Yaskawa INFORM job: BATMAN_2STR.JBI

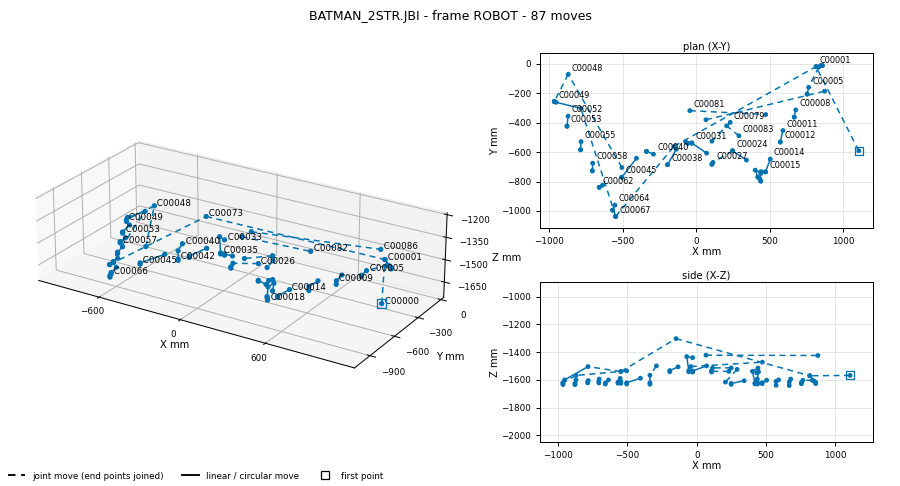
[picture p0: tool path of BATMAN_2STR.JBI in frame ROBOT, 87 of 158 moves have a stored position in this frame; points joined in program order, loops and branches not executed]
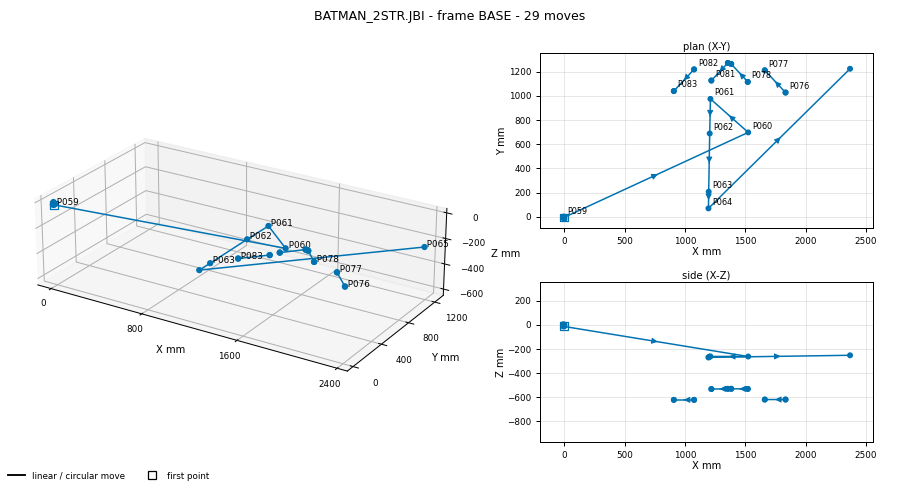
[picture p1: tool path of BATMAN_2STR.JBI in frame BASE, 29 of 158 moves have a stored position in this frame; points joined in program order, loops and branches not executed]
/JOB
//NAME BATMAN_2STR
///FOLDERNAME KRIS-SCIANA
//POS
///NPOS 87,87,0,38,0,0
///TOOL 0
///POSTYPE ROBOT
///RECTAN
///RCONF 0,0,0,0,0,0,0,0,0,0,0,0,0,0,0,0,0,0,0,0,0,0,0,0
C00000=1105.156,-590.615,-1567.354,6.0584,32.6468,147.4704
C00001=815.315,-18.001,-1569.939,-1.7381,27.7880,143.5527
C00002=857.710,-10.973,-1618.417,-1.7378,27.7886,143.5541
C00003=857.707,-10.971,-1626.567,-1.7382,27.7883,143.5526
C00004=833.675,-21.061,-1602.919,-1.7360,27.7873,143.5574
C00005=764.713,-159.460,-1602.917,-1.7360,27.7871,143.5577
C00006=754.333,-205.391,-1618.911,-1.7368,27.7882,143.5563
C00007=754.360,-205.381,-1627.221,-1.7390,27.7891,143.5536
C00008=676.929,-312.752,-1594.094,-1.7387,27.7900,143.5534
C00009=666.860,-361.337,-1616.296,-1.7391,27.7907,143.5606
C00010=666.607,-362.154,-1640.305,-1.7382,27.7861,143.5578
C00011=589.702,-453.220,-1599.704,-1.7386,27.7882,143.5565
C00012=571.550,-531.474,-1610.685,-1.7384,27.7889,143.5556
C00013=571.577,-531.526,-1638.417,-1.7371,27.7932,143.5506
C00014=503.343,-647.565,-1602.574,-1.7244,27.7369,143.5385
C00015=471.201,-734.222,-1620.126,-1.7395,27.7918,143.5502
C00016=471.196,-734.208,-1626.856,-1.7400,27.7912,143.5505
C00017=439.050,-796.935,-1621.095,-1.7408,27.7924,143.5517
C00018=439.049,-796.953,-1629.727,-1.7399,27.7928,143.5504
C00019=441.123,-742.830,-1514.057,-1.7418,27.7901,143.5526
C00020=401.170,-722.445,-1537.720,10.1454,37.8099,55.1563
C00021=419.273,-769.804,-1621.635,10.0244,37.5346,56.2633
C00022=419.267,-769.795,-1628.682,10.0249,37.5342,56.2644
C00023=341.517,-653.963,-1605.800,10.0246,37.5341,56.2657
C00024=247.787,-591.524,-1625.473,10.0271,37.5316,56.2731
C00025=247.794,-591.522,-1631.709,10.0263,37.5313,56.2715
C00026=247.796,-591.525,-1513.148,10.0256,37.5315,56.2705
C00027=113.704,-669.750,-1513.152,10.0280,37.5312,56.2733
C00028=106.856,-682.927,-1533.943,10.0224,37.5325,56.2697
C00029=106.874,-682.958,-1542.733,10.0189,37.5339,56.2663
C00030=70.694,-606.931,-1498.730,10.0200,37.5334,56.2633
C00031=-30.272,-538.287,-1535.198,10.0214,37.5337,56.2637
C00032=-30.275,-538.292,-1543.514,10.0219,37.5340,56.2653
C00033=-30.277,-538.270,-1439.519,10.0239,37.5323,56.2676
C00034=-72.212,-529.493,-1431.848,10.0246,37.5336,126.4601
C00035=-58.288,-539.735,-1534.232,10.0230,37.5329,126.4597
C00036=-58.298,-539.747,-1541.111,10.0251,37.5325,126.4632
C00037=-134.942,-579.910,-1505.733,10.0214,37.5335,126.4526
C00038=-194.951,-685.626,-1532.619,10.0192,37.5313,126.4507
C00039=-194.945,-685.631,-1541.099,10.0183,37.5324,126.4483
C00040=-291.274,-613.943,-1498.709,10.0193,37.5315,126.4500
C00041=-338.146,-594.905,-1566.079,10.0206,37.5306,126.4559
C00042=-338.153,-594.908,-1620.637,10.0213,37.5304,126.4568
C00043=-338.152,-594.897,-1631.211,10.0213,37.5296,126.4575
C00044=-406.496,-641.674,-1587.377,10.0204,37.5303,126.4602
C00045=-505.818,-770.602,-1620.991,10.0161,37.5294,126.4561
C00046=-505.822,-770.602,-1629.641,10.0170,37.5289,126.4582
C00047=-505.818,-704.683,-1534.604,10.0172,37.5293,126.4596
C00048=-870.558,-70.607,-1567.754,-5.5732,23.9550,-0.0620
C00049=-965.415,-255.754,-1620.582,-3.4263,30.0338,0.8210
C00050=-965.418,-255.752,-1622.018,-3.4258,30.0337,0.8220
C00051=-965.421,-255.747,-1633.054,-3.4254,30.0337,0.8221
C00052=-871.675,-355.111,-1600.349,-3.4260,30.0340,0.8216
C00053=-878.724,-423.891,-1625.207,-3.4243,30.0345,0.8253
C00054=-878.718,-423.902,-1634.168,-3.4261,30.0338,0.8213
C00055=-782.869,-528.764,-1604.816,-3.4248,30.0318,0.8156
C00056=-786.737,-583.960,-1612.292,-3.4246,30.0303,0.8183
C00057=-786.740,-583.966,-1621.129,-3.4247,30.0307,0.8203
C00058=-704.142,-675.428,-1593.875,-3.4274,30.0320,0.8194
C00059=-706.471,-727.273,-1611.725,-3.4351,30.0238,0.8165
C00060=-706.461,-727.277,-1621.357,-3.4355,30.0231,0.8168
C00061=-637.422,-825.106,-1600.424,-3.4351,30.0208,0.8167
C00062=-659.834,-839.485,-1622.110,-3.4334,30.0214,0.8205
C00063=-659.844,-839.500,-1629.778,-3.4344,30.0221,0.8200
C00064=-552.859,-959.979,-1588.724,-3.4350,30.0244,0.8136
C00065=-568.518,-994.720,-1614.958,-3.4362,30.0232,0.8143
C00066=-568.514,-994.724,-1623.430,-3.4363,30.0225,0.8125
C00067=-547.865,-1036.819,-1613.327,-3.4355,30.0239,0.8160
C00068=-547.869,-1036.811,-1624.522,-3.4350,30.0238,0.8135
C00069=-547.867,-1036.815,-1539.725,-3.4353,30.0236,0.8134
C00070=-784.559,-302.239,-1503.879,-3.4366,30.0265,0.8087
C00071=-953.024,-261.100,-1599.401,-3.4345,30.0250,0.8092
C00072=-547.867,-1036.815,-1539.725,-3.4353,30.0236,0.8134
C00073=-149.962,-559.854,-1302.120,-3.4346,30.0247,0.8146
C00074=815.315,-18.001,-1569.939,-1.7381,27.7880,143.5527
C00075=847.137,-11.115,-1608.986,-1.7371,27.7876,143.5542
C00076=432.100,-781.158,-1548.511,-1.7395,27.7865,143.5518
C00077=445.125,-733.631,-1540.567,-2.7194,23.4640,36.3665
C00078=436.491,-734.622,-1593.359,-2.7195,23.4653,36.3724
C00079=231.186,-397.551,-1538.170,10.0369,37.5564,56.2933
C00080=106.565,-525.549,-1538.164,10.0364,37.5570,56.2931
C00081=-43.468,-317.794,-1503.609,10.0906,37.0928,60.8768
C00082=472.745,-344.262,-1471.900,21.7977,37.1280,159.9819
C00083=290.461,-488.573,-1524.026,10.0019,37.5312,126.4207
C00084=206.735,-421.024,-1615.254,10.0028,37.5295,126.4201
C00085=66.048,-379.716,-1421.439,10.0175,37.5426,126.4581
C00086=873.206,-185.580,-1423.876,-1.7383,27.7862,-167.3950
BC00000=938.923,1838.231,1681.523
BC00001=1421.588,1829.899,1010.263
BC00002=1421.588,1829.899,1010.263
BC00003=1421.588,1829.899,1010.263
BC00004=1421.581,1829.905,1010.257
BC00005=1421.581,1829.905,1010.257
BC00006=1421.581,1829.905,1010.257
BC00007=1421.581,1829.905,1010.257
BC00008=1421.581,1829.905,1010.257
BC00009=1421.581,1829.905,1010.257
BC00010=1421.581,1829.905,1010.257
BC00011=1421.581,1829.905,1010.257
BC00012=1421.581,1829.905,1010.257
BC00013=1421.581,1829.905,1010.257
BC00014=1421.581,1829.905,1010.257
BC00015=1421.581,1829.905,1010.257
BC00016=1421.581,1829.905,1010.257
BC00017=1421.581,1829.905,1010.257
BC00018=1421.581,1829.905,1010.257
BC00019=1421.581,1829.905,1010.254
BC00020=1421.581,1829.912,1010.248
BC00021=1414.141,1827.243,1016.162
BC00022=1414.141,1827.243,1016.162
BC00023=1414.141,1827.243,1016.162
BC00024=1414.141,1827.243,1016.162
BC00025=1414.141,1827.243,1016.162
BC00026=1414.141,1827.243,1016.162
BC00027=1414.141,1827.243,1016.162
BC00028=1414.141,1827.243,1016.162
BC00029=1414.141,1827.243,1016.162
BC00030=1414.141,1827.243,1016.162
BC00031=1414.141,1827.243,1016.162
BC00032=1414.141,1827.243,1016.162
BC00033=1414.141,1827.243,1016.162
BC00034=1414.141,1827.243,1016.162
BC00035=1414.141,1827.243,1016.162
BC00036=1414.141,1827.243,1016.162
BC00037=1414.141,1827.243,1016.162
BC00038=1414.141,1827.243,1016.162
BC00039=1414.141,1827.243,1016.162
BC00040=1414.141,1827.243,1016.162
BC00041=1414.141,1827.243,1016.162
BC00042=1414.141,1827.243,1016.162
BC00043=1414.141,1827.243,1016.162
BC00044=1414.141,1827.243,1016.162
BC00045=1414.141,1827.243,1016.162
BC00046=1414.141,1827.243,1016.162
BC00047=1414.141,1827.243,1016.162
BC00048=1421.581,1829.905,1010.254
BC00049=1421.581,2077.513,1010.254
BC00050=1421.581,2077.513,1010.254
BC00051=1421.581,2077.513,1010.254
BC00052=1421.581,2077.513,1010.248
BC00053=1421.581,2077.513,1010.248
BC00054=1421.581,2077.513,1010.248
BC00055=1421.581,2077.513,1010.248
BC00056=1421.581,2077.513,1010.248
BC00057=1421.581,2077.513,1010.248
BC00058=1421.581,2077.513,1010.248
BC00059=1421.581,2077.507,1010.244
BC00060=1421.581,2077.507,1010.244
BC00061=1421.581,2077.507,1010.244
BC00062=1421.581,2077.507,1010.244
BC00063=1421.581,2077.507,1010.244
BC00064=1421.581,2077.507,1010.244
BC00065=1421.581,2077.507,1010.244
BC00066=1421.581,2077.507,1010.244
BC00067=1421.581,2077.507,1010.244
BC00068=1421.581,2077.507,1010.244
BC00069=1421.581,2077.507,1010.244
BC00070=1421.581,2077.507,1010.244
BC00071=1421.581,2077.507,1010.244
BC00072=1421.581,2077.507,1010.244
BC00073=1421.581,2077.507,1010.244
BC00074=1421.588,1829.899,1010.263
BC00075=1421.588,1829.899,1010.263
BC00076=1421.588,1829.899,1010.263
BC00077=1421.588,1829.899,1010.263
BC00078=1421.588,1829.899,1010.263
BC00079=1436.938,1677.545,1031.627
BC00080=1436.938,1677.545,1031.627
BC00081=1441.270,1634.546,1037.657
BC00082=838.758,1634.546,1037.657
BC00083=842.369,1626.975,1038.719
BC00084=842.369,1626.975,1038.719
BC00085=842.362,1626.982,1038.713
BC00086=845.778,2972.171,1682.637
///POSTYPE BASE
P00059=-2.448,-6.714,-12.718,0.0000,0.0000,0.0000
P00060=1524.284,698.404,-261.973,-0.4635,36.8346,-1.2388
P00061=1211.499,975.999,-261.374,0.5148,35.2356,175.5099
P00062=1205.574,689.500,-262.704,0.5159,35.2461,175.5270
P00063=1197.217,207.358,-268.729,0.4863,35.2395,175.4586
P00064=1195.199,68.975,-269.171,0.5092,35.2366,175.4908
P00065=2367.684,1225.356,-251.745,0.6375,35.5356,-175.5535
P00070=2.449,-18.318,2.615,0.0000,0.0000,0.0000
P00071=-2.048,-0.034,-9.092,0.0000,0.0000,0.0000
P00072=-1.595,-0.049,-6.373,0.0000,0.0000,0.0000
P00073=-8.474,-10.331,-11.894,0.0000,0.0000,0.0000
P00074=1.731,-3.007,-10.460,0.0000,0.0000,0.0000
///RCONF 0,1,0,0,0,0,0,0,0,0,0,0,0,0,0,0,0,0,0,0,0,0,0,0
P00075=-9.634,0.014,4.922,0.0000,0.0000,0.0000
///RCONF 0,0,0,0,0,0,0,0,0,0,0,0,0,0,0,0,0,0,0,0,0,0,0,0
P00076=1833.500,1028.615,-618.215,10.0256,37.5190,56.2681
P00077=1661.766,1212.555,-618.325,10.0309,37.5577,56.2858
P00078=1520.740,1116.757,-530.271,10.0398,37.5578,56.2925
P00079=1383.754,1265.334,-529.217,10.0293,37.5461,56.2787
P00080=1355.833,1273.708,-529.583,10.0283,37.5305,126.4716
P00081=1219.184,1127.874,-531.327,10.0137,37.5345,126.4324
P00082=1075.995,1220.294,-620.895,10.0203,37.5289,126.4576
P00083=908.434,1040.970,-620.895,10.0141,37.5419,126.4584
P00087=-17.000,-22.000,-3.000,0.0000,0.0000,0.0000
P00088=-8.588,-0.108,-11.097,0.0000,0.0000,0.0000
P00089=5.931,-12.286,-8.772,0.0000,0.0000,0.0000
P00090=-14.057,13.261,-6.464,0.0000,0.0000,0.0000
P00091=1.048,0.648,3.624,0.0000,0.0000,0.0000
P00092=12.000,-9.000,-4.000,0.0000,0.0000,0.0000
P00093=-12.000,12.000,-3.000,0.0000,0.0000,0.0000
P00094=10.000,10.000,-3.000,0.0000,0.0000,0.0000
P00095=-11.943,-14.820,-6.815,0.0000,0.0000,0.0000
P00096=-4.844,-19.262,-10.890,0.0000,0.0000,0.0000
P00108=0.000,0.000,-3.000,0.0000,0.0000,0.0000
P00123=0.000,-50.000,0.000,0.0000,0.0000,0.0000
P00125=0.000,0.000,2.400,0.0000,0.0000,0.0000
P00126=-50.000,0.000,0.000,0.0000,0.0000,0.0000
P00127=50.000,0.000,0.000,0.0000,0.0000,0.0000
P00172=2.000,-12.000,-3.000,0.0000,0.0000,40.0000
P00173=-5.000,-9.000,-2.400,0.0000,0.0000,-15.0000
//INST
///DATE 2024/05/06 12:47
///COMM NOWY SEARCH
///ATTR SC,RW,RJ
////FRAME ROBOT
///GROUP1 RB1,BS1
NOP
SFTOF
MOVJ C00000 BC00000 VJ=60.00
MOVJ C00001 BC00001 VJ=60.00
'POMIAR PRAWA STRONA
'1
MOVL C00002 BC00002 V=166.7
MOVL C00003 BC00003 V=16.7 PL=0 SRCH RIN#(1)=ON T=1.00 DIS=20.0
TIMER T=0.20
IMOV P125 V=13.3 PL=0
TIMER T=0.20
IMOV P127 V=13.3 PL=0 SRCH RIN#(1)=ON DIS=20.0
TIMER T=0.20
GETS PX070 $PX001
TIMER T=0.10
MOVJ C00004 BC00004 VJ=15.00
MOVJ C00005 BC00005 VJ=15.00
'2
MOVL C00006 BC00006 V=50.0
MOVL C00007 BC00007 V=16.7 PL=0 SRCH RIN#(1)=ON T=1.00 DIS=20.0
TIMER T=0.20
IMOV P125 V=13.3 PL=0
TIMER T=0.20
IMOV P127 V=13.3 PL=0 SRCH RIN#(1)=ON DIS=20.0
TIMER T=0.20
GETS PX071 $PX001
TIMER T=0.10
MOVJ C00008 BC00008 VJ=15.00
'3
MOVL C00009 BC00009 V=50.0
MOVL C00010 BC00010 V=16.7 PL=0 SRCH RIN#(1)=ON T=1.00 DIS=20.0
TIMER T=0.20
IMOV P125 V=13.3 PL=0
TIMER T=0.20
IMOV P127 V=13.3 PL=0 SRCH RIN#(1)=ON DIS=20.0
TIMER T=0.20
GETS PX072 $PX001
TIMER T=0.10
MOVJ C00011 BC00011 VJ=15.00
'4
MOVL C00012 BC00012 V=50.0
MOVL C00013 BC00013 V=16.7 PL=0 SRCH RIN#(1)=ON T=1.00 DIS=20.0
TIMER T=0.20
IMOV P125 V=13.3 PL=0
TIMER T=0.20
IMOV P127 V=13.3 PL=0 SRCH RIN#(1)=ON DIS=20.0
TIMER T=0.20
GETS PX073 $PX001
TIMER T=0.10
MOVJ C00014 BC00014 VJ=15.00
'5
MOVL C00015 BC00015 V=50.0
MOVL C00016 BC00016 V=16.7 PL=0 SRCH RIN#(1)=ON T=1.00 DIS=20.0
TIMER T=0.20
IMOV P125 V=13.3 PL=0
TIMER T=0.20
IMOV P127 V=13.3 PL=0 SRCH RIN#(1)=ON DIS=20.0
TIMER T=0.20
GETS PX074 $PX001
TIMER T=0.10
MOVL C00017 BC00017 V=50.0
MOVL C00018 BC00018 V=16.7 PL=0 SRCH RIN#(1)=ON T=1.00 DIS=20.0
TIMER T=0.20
IMOV P125 V=13.3 PL=0
TIMER T=0.20
IMOV P127 V=13.3 PL=0 SRCH RIN#(1)=ON DIS=20.0
TIMER T=0.20
GETS PX075 $PX001
TIMER T=0.10
MOVJ C00019 BC00019 VJ=15.00
MOVJ C00020 BC00020 VJ=30.00
'POMIAR BATMAN
MOVL C00021 BC00021 V=166.7
MOVL C00022 BC00022 V=16.7 PL=0 SRCH RIN#(1)=ON T=1.00 DIS=20.0
TIMER T=0.20
IMOV P125 V=13.3 PL=0
TIMER T=0.20
IMOV P123 V=13.3 PL=0 SRCH RIN#(1)=ON DIS=20.0
TIMER T=0.20
GETS PX076 $PX001
TIMER T=0.10
MOVJ C00023 BC00023 VJ=30.00
MOVL C00024 BC00024 V=166.7
MOVL C00025 BC00025 V=16.7 PL=0 SRCH RIN#(1)=ON T=1.00 DIS=20.0
TIMER T=0.20
IMOV P125 V=13.3 PL=0
TIMER T=0.20
IMOV P123 V=13.3 PL=0 SRCH RIN#(1)=ON DIS=20.0
TIMER T=0.20
GETS PX077 $PX001
TIMER T=0.10
MOVJ C00026 BC00026 VJ=30.00
MOVJ C00027 BC00027 VJ=30.00
MOVL C00028 BC00028 V=166.7
MOVL C00029 BC00029 V=16.7 PL=0 SRCH RIN#(1)=ON T=1.00 DIS=20.0
TIMER T=0.20
IMOV P125 V=13.3 PL=0
TIMER T=0.20
IMOV P123 V=13.3 PL=0 SRCH RIN#(1)=ON DIS=20.0
TIMER T=0.20
GETS PX078 $PX001
TIMER T=0.10
MOVJ C00030 BC00030 VJ=30.00
MOVL C00031 BC00031 V=166.7
MOVL C00032 BC00032 V=16.7 PL=0 SRCH RIN#(1)=ON T=1.00 DIS=20.0
TIMER T=0.20
IMOV P125 V=13.3 PL=0
TIMER T=0.20
IMOV P123 V=13.3 PL=0 SRCH RIN#(1)=ON DIS=20.0
TIMER T=0.20
GETS PX079 $PX001
TIMER T=0.10
MOVJ C00033 BC00033 VJ=30.00
MOVJ C00034 BC00034 VJ=30.00
MOVL C00035 BC00035 V=166.7
MOVL C00036 BC00036 V=16.7 PL=0 SRCH RIN#(1)=ON T=1.00 DIS=20.0
TIMER T=0.20
IMOV P125 V=13.3 PL=0
TIMER T=0.20
IMOV P123 V=13.3 PL=0 SRCH RIN#(1)=ON DIS=20.0
TIMER T=0.20
GETS PX080 $PX001
TIMER T=0.10
MOVJ C00037 BC00037 VJ=30.00
MOVL C00038 BC00038 V=166.7
MOVL C00039 BC00039 V=16.7 PL=0 SRCH RIN#(1)=ON T=1.00 DIS=20.0
TIMER T=0.20
IMOV P125 V=13.3 PL=0
TIMER T=0.20
IMOV P123 V=13.3 PL=0 SRCH RIN#(1)=ON DIS=20.0
TIMER T=0.20
GETS PX081 $PX001
TIMER T=0.10
MOVJ C00040 BC00040 VJ=30.00
MOVJ C00041 BC00041 VJ=30.00
MOVL C00042 BC00042 V=166.7
MOVL C00043 BC00043 V=16.7 PL=0 SRCH RIN#(1)=ON T=1.00 DIS=20.0
TIMER T=0.20
IMOV P125 V=13.3 PL=0
TIMER T=0.20
IMOV P123 V=13.3 PL=0 SRCH RIN#(1)=ON DIS=20.0
TIMER T=0.20
GETS PX082 $PX001
TIMER T=0.10
MOVJ C00044 BC00044 VJ=30.00
MOVL C00045 BC00045 V=166.7
MOVL C00046 BC00046 V=16.7 PL=0 SRCH RIN#(1)=ON T=1.00 DIS=20.0
TIMER T=0.20
IMOV P125 V=13.3 PL=0
TIMER T=0.20
IMOV P123 V=13.3 PL=0 SRCH RIN#(1)=ON DIS=20.0
TIMER T=0.20
GETS PX083 $PX001
TIMER T=0.10
MOVJ C00047 BC00047 VJ=30.00
'KONIEC POMIAR BATMAN 1STR
SFTOF
MOVJ C00048 BC00048 VJ=50.00
SFTOF
MOVJ C00049 BC00049 VJ=15.00
'1
MOVL C00050 BC00050 V=166.7
MOVL C00051 BC00051 V=16.7 PL=0 SRCH RIN#(1)=ON T=1.00 DIS=20.0
TIMER T=0.20
IMOV P125 V=13.3 PL=0
TIMER T=0.20
IMOV P126 V=13.3 PL=0 SRCH RIN#(1)=ON DIS=20.0
TIMER T=0.20
GETS PX059 $PX001
TIMER T=0.10
MOVJ C00052 BC00052 VJ=15.00
MOVL C00053 BC00053 V=166.7
MOVL C00054 BC00054 V=16.7 PL=0 SRCH RIN#(1)=ON T=1.00 DIS=20.0
TIMER T=0.20
IMOV P125 V=13.3 PL=0
TIMER T=0.20
IMOV P126 V=13.3 PL=0 SRCH RIN#(1)=ON DIS=20.0
TIMER T=0.20
GETS PX060 $PX001
TIMER T=0.10
MOVJ C00055 BC00055 VJ=50.00
'2
MOVL C00056 BC00056 V=50.0
MOVL C00057 BC00057 V=16.7 PL=0 SRCH RIN#(1)=ON T=1.00 DIS=30.0
TIMER T=0.20
IMOV P125 V=13.3 PL=0
TIMER T=0.20
IMOV P126 V=13.3 PL=0 SRCH RIN#(1)=ON DIS=20.0
TIMER T=0.20
GETS PX061 $PX001
TIMER T=0.10
MOVJ C00058 BC00058 VJ=50.00
'3
MOVL C00059 BC00059 V=50.0
MOVL C00060 BC00060 V=16.7 PL=0 SRCH RIN#(1)=ON T=1.00 DIS=30.0
TIMER T=0.20
IMOV P125 V=13.3 PL=0
TIMER T=0.20
IMOV P126 V=13.3 PL=0 SRCH RIN#(1)=ON DIS=20.0
TIMER T=0.20
GETS PX062 $PX001
TIMER T=0.10
MOVJ C00061 BC00061 VJ=50.00
'4
MOVL C00062 BC00062 V=50.0
MOVL C00063 BC00063 V=16.7 PL=0 SRCH RIN#(1)=ON T=1.00 DIS=30.0
TIMER T=0.20
IMOV P125 V=13.3 PL=0
TIMER T=0.20
IMOV P126 V=13.3 PL=0 SRCH RIN#(1)=ON DIS=20.0
TIMER T=0.20
GETS PX063 $PX001
TIMER T=0.10
MOVJ C00064 BC00064 VJ=15.00
'5
MOVL C00065 BC00065 V=50.0
MOVL C00066 BC00066 V=16.7 PL=0 SRCH RIN#(1)=ON T=1.00 DIS=20.0
TIMER T=0.20
IMOV P125 V=13.3 PL=0
TIMER T=0.20
IMOV P126 V=13.3 PL=0 SRCH RIN#(1)=ON DIS=20.0
TIMER T=0.20
GETS PX064 $PX001
TIMER T=0.10
MOVL C00067 BC00067 V=50.0
MOVL C00068 BC00068 V=16.7 PL=0 SRCH RIN#(1)=ON T=1.00 DIS=20.0
TIMER T=0.20
IMOV P125 V=13.3 PL=0
TIMER T=0.20
IMOV P126 V=13.3 PL=0 SRCH RIN#(1)=ON DIS=20.0
TIMER T=0.20
GETS PX065 $PX001
TIMER T=0.10
MOVJ C00069 BC00069 VJ=15.00
'********
'********
'********
MOVJ C00070 BC00070 VJ=15.00
MOVL C00071 BC00071 V=333.3
MACRO1 MJ#(0) ARGF7
SFTOF
SFTON P095
MOVL P059 V=83.3
ARCON
MOVL P060 V=10.8
MOVL P061 V=10.8
ARCON
MOVL P062 V=10.8
MOVL P063 V=10.8
MOVL P064 V=10.8
SFTOF
SFTON P172
MOVL P065 V=10.8
ARCOF
MOVJ C00072 BC00072 VJ=15.00
SFTOF
MOVJ C00073 BC00073 VJ=15.00
MOVJ C00074 BC00074 VJ=40.00
SFTON P096
MOVJ C00075 BC00075 VJ=15.00
MOVL P070 V=83.3
ARCON
MOVL P071 V=10.8
MOVL P072 V=10.8
MOVL P073 V=10.8
MOVL P074 V=10.8
SFTOF
SFTON P173
MOVL P075 V=10.8
ARCOF
SFTOF
MOVJ C00076 BC00076 VJ=15.00
MOVJ C00077 BC00077 VJ=30.00
'START SPAWANIE BATMAN
MOVJ C00078 BC00078 VJ=30.00
SFTON P090
MOVL P076 V=83.3
SFTOF
ARCON
SFTON P108
ARCON
MOVL P076 V=10.8
MOVL P077 V=10.8
SFTOF
SFTON P091
MOVL P077 V=10.8
ARCOF
SFTOF
MOVJ C00079 BC00079 VJ=30.00
MOVJ C00080 BC00080 VJ=30.00
SFTON P092
MOVL P078 V=83.3
ARCON
SFTOF
SFTON P108
MOVL P078 V=10.8
MOVL P079 V=10.8
SFTOF
SFTON P093
MOVL P079 V=10.8
ARCOF
SFTOF
MOVJ C00081 BC00081 VJ=30.00
MOVJ C00082 BC00082 VJ=30.00
SFTON P094
MOVL P080 V=83.3
SFTOF
ARCON
SFTON P108
MOVL P080 V=10.8
MOVL P081 V=10.8
SFTOF
SFTON P087
MOVL P081 V=10.8
SFTOF
ARCOF
MOVJ C00083 BC00083 VJ=30.00
MOVJ C00084 BC00084 VJ=30.00
SFTON P088
MOVL P082 V=83.3
SFTOF
ARCON
SFTON P108
MOVL P082 V=10.8
MOVL P083 V=10.8
SFTOF
SFTON P089
MOVL P083 V=10.8
SFTOF
ARCOF
MOVJ C00085 BC00085 VJ=30.00
MOVJ C00086 BC00086 VJ=100.00
CALL JOB:ONLYCUT-R1_LONG
END
